{attribute 'GeneratedUsingTerminal: EP3182-1002-0017'}
{attribute addProperty BoxType "EP3182-1002-0017"}
{attribute addProperty Id "AI_Standard_Channel_1AT %I*AI_Standard_Channel_4A3944819AI_Standard_Channel_2AT %I*AI_Standard_Channel_4A3944819DO_OutputsAT %Q*DO_Outputs_C0F4C3832WcStateAT %I*WcState_9091E0EB2InfoDataAT %I*InfoData_32EB74EA10"}
{attribute addProperty CRC "198275543"}
{attribute addProperty Size "32"}
TYPE EP3182_0BD171D7 EXTENDS EtcSlaveTerminalBase_947E5A46 :
STRUCT
	{attribute addProperty Name "AI_Standard_Channel_1"}
	AI_Standard_Channel_1 : AI_Standard_Channel_4A394481;
	{attribute addProperty Name "AI_Standard_Channel_2"}
	AI_Standard_Channel_2 : AI_Standard_Channel_4A394481;
	{attribute addProperty Name "DO_Outputs"}
	DO_Outputs : DO_Outputs_C0F4C383;
	{attribute addProperty Name "WcState"}
	WcState : WcState_9091E0EB;
	{attribute addProperty Name "InfoData"}
	InfoData : InfoData_32EB74EA;
END_STRUCT
END_TYPE

(* stored: Version 1.2.0.0, ProductVersion 3.1.4024.9
   DUT EP3182_0BD171D7: Id {48ab1101-1d5f-4dd6-ae98-91a43e8d762a} *)
